// TIA Portal V16 export
// export: Created 2023-03-29T11:03:44.7031176Z, ExportSetting WithDefaults, DisplayName Totally Integrated Automation Portal, DisplayVersion V16 Update 6, DisplayName TIA Portal Version Control Interface, DisplayVersion V16 Update 2, DisplayName TIA Portal Openness, DisplayVersion V16 Update 6, DisplayName STEP 7 Professional, DisplayVersion V16 Update 6, DisplayName STEP 7 Safety, DisplayVersion V16, DisplayName WinCC Advanced, DisplayVersion V16 Update 6
VAR_GLOBAL   // PLC tag table "Z2"
   Hbit_Reset_Z2 AT %M12.6 : Bool;
   inputREMT_Z_2 AT %M53.1 : Bool;   // znacznik wejście zdalne
   Hbit_Zamknij_Z2 AT %M12.5 : Bool;
   Hbit_Otwarta_Z2 AT %M12.1 : Bool;
   Byte_Status_Z2 AT %MW12 : Word;   // Słowo statusu napędu
   inputAwariaMomentZ_2 AT %M53.5 : Bool;   // znacznik wejście
   inputZamkniętaZ_2 AT %M53.3 : Bool;   // znacznik wejście
   Hbit_Alarm_Z2 AT %M12.0 : Bool;
   Hbit_Zamknieta_Z2 AT %M12.3 : Bool;
   inputRuch_Z_2 AT %M53.4 : Bool;
   setSVMC_Z_2 AT %M54.3 : Bool;   // Znacznik polecenia zamknij w trybie automat
   inputAumalokalneZ_2 AT %M53.6 : Bool;   // znacznik wejście
   Hbit_Auto_Manu_Z2 AT %M12.7 : Bool;
   Hbit_Otwórz_Z2 AT %M12.4 : Bool;
   CMD_Open_Z_2 AT %M54.5 : Bool;   // załącz otwieranie
   inputAumaawariaZ_2 AT %M54.1 : Bool;   // znacznik wejście
   Hbit_REN_Z2 AT %M12.2 : Bool;
   isAUMA_Z_2 AT %M44.0 : Bool;   // przęłącznik wymiany na AUMA
   inputAumaautomatZ_2 AT %M53.7 : Bool;   // znacznik wejście
   setAlarm_Moment_Z_2 AT %M54.4 : Bool;   // znacznik alarmu od momentówki w trybie zdalnym (aut/mamnual)
   setSVMO_Z_2 AT %M54.2 : Bool;   // Znacznik polecenia otwórz w trybie automat
   isGotowość_Z_2 AT %M53.0 : Bool;   // bit gotowości wspólny
   inputOtwartaZ_2 AT %M53.2 : Bool;   // znacznik wejście
   CMD_Awaria_Z_2 AT %M54.7 : Bool;   // Awaria zbiorcza
   CMD_Close_Z_2 AT %M54.6 : Bool;   // załącz zamykanie
   inputAumagotowośćZ_2 AT %M54.0 : Bool;   // znacznik wejście
   edge_Hz_Z2 AT %M92.0 : Bool;   // pamięć zbocza 1 Hz
END_VAR
